FUNCTION_BLOCK FB_MappingOutputs
VAR_INPUT
END_VAR
VAR_OUTPUT
END_VAR
VAR
END_VAR

// Exercice 1
FIO_Output1[0] := FIO_O_VoyantMarche;
FIO_Output1[1] := FIO_O_Convoyeur;
FIO_Output1[2] := FIO_O_VoyantAvancer;

END_FUNCTION_BLOCK

(* stored: Version 1.1.0.1, ProductVersion 3.1.4024.11
   POU FB_MappingOutputs: Id {7837aa2e-7999-4e5c-9130-5f0d63f85a7a}, SpecialFunc None *)
